# EPICS autosave request: support/love/3-2-4/loveApp/Db/Love_settings.req
# Love controller
$(P)$(Q)Disable.VAL
$(P)$(Q)FastFanout.SCAN
$(P)$(Q)SlowFanout.SCAN
$(P)$(Q)PutSetPt1.VAL
$(P)$(Q)PutSetPt2.VAL
$(P)$(Q)PutAlarmLo.VAL
$(P)$(Q)PutAlarmHi.VAL
$(P)$(Q)Value.DESC
